FUNCTION_BLOCK SELECT_MODE
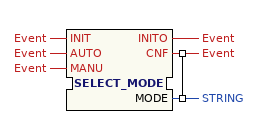
  EVENT_INPUT
    INIT;
    AUTO;
    MANU;
  END_EVENT
  EVENT_OUTPUT
    INITO;
    CNF WITH MODE;
  END_EVENT
  VAR_OUTPUT
    MODE : STRING;
  END_VAR
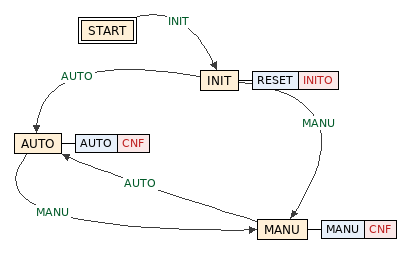
  EC_STATES
    START;
    AUTO : AUTO -> CNF;
    MANU : MANU -> CNF;
    INIT : RESET -> INITO;
  END_STATES
  EC_TRANSITIONS
    INIT TO AUTO := AUTO;
    INIT TO MANU := MANU;
    AUTO TO MANU := MANU;
    MANU TO AUTO := AUTO;
    START TO INIT := INIT;
  END_TRANSITIONS
  ALGORITHM AUTO IN ST:
MODE := &#39;AUTO&#39;;&#38;#10;
  END_ALGORITHM
  ALGORITHM MANU IN ST:
MODE := &#39;MANU&#39;;&#38;#10;
  END_ALGORITHM
  ALGORITHM RESET IN ST:
MODE := &#39;&#39;;&#38;#10;
  END_ALGORITHM
END_FUNCTION_BLOCK
